INTERFACE INTERNAL I_SignalNode EXTENDS I_Debug

PROPERTY INTERNAL _End : UDINT
GET
END_GET
SET
END_SET
END_PROPERTY

PROPERTY INTERNAL _Id : UDINT
GET
END_GET
END_PROPERTY

PROPERTY INTERNAL _Size : UDINT
GET
END_GET
SET
END_SET
END_PROPERTY

PROPERTY INTERNAL _Start : UDINT
GET
END_GET
SET
END_SET
END_PROPERTY

END_INTERFACE

(* stored: Version 1.1.0.1
   Itf I_SignalNode: Id {9986a83b-84ba-44f5-ada8-fdbfebb0d1eb}
   Folder _: Id {2c045e55-1443-473c-b9f7-83217e57ae9d}
   Property _End: Id {3e24d41f-d222-4c9c-bf00-72565b4682aa}
   Get Get: Id {a849bc8e-3624-4b20-a478-b5ecdef96a27}
   Set Set: Id {f6497037-d1b8-4c02-aea9-dc377a107f68}
   Property _Id: Id {a9792a04-1aee-40d0-8866-c6ab68d00823}
   Get Get: Id {76d7e66f-9343-4a9b-8c42-82219155ae4d}
   Property _Size: Id {b6650d71-cbcf-43b0-88e5-bb4cde5396b4}
   Get Get: Id {babf9e29-0594-4bde-8bfe-731925a65630}
   Set Set: Id {dd2179e8-aeab-4379-b8dc-bfc944182c00}
   Property _Start: Id {30a15fd0-e880-4534-8545-dc470cc15d81}
   Get Get: Id {692bd17a-bf66-4c05-9a36-ebed70b02fe3}
   Set Set: Id {9a03a416-271a-4300-ab9a-b087a7d84576} *)
